INTERFACE I_Action

METHOD Perform
VAR_INPUT
    performCaseNumber : INT;
END_VAR
VAR_IN_OUT
    item : POINTER TO Object;
END_VAR
END_METHOD

END_INTERFACE

(* stored: Version 1.1.0.1, ProductVersion 3.1.4024.6
   Itf I_Action: Id {cead35ff-aed5-4b3d-b8fd-4c4da36ec2ee}
   Method Perform: Id {649842f8-9bac-478c-9416-f22fb18098e2} *)
